IF _bIsFirstSeg AND _bIsLastSeg THEN	
	_sPath := '';
    _nLen := 0;
	_nSegStart := 0;
	_nSegEnd := 0;
	RemoveAndNext := Ok;
ELSIF _bIsFirstSeg THEN
	_sPath := Tc2_Standard.DELETE(_sPath, _nSegLen + 1, _nSegStart); // Also removes dot after first segment
	_nLen := _nLen - _nSegLen;
	_nSegStart := 0;
	_nSegEnd := 0;
	RemoveAndNext := Ok;
ELSIF _bIsLastSeg THEN
	_sPath := Tc2_Standard.DELETE(_sPath, _nSegLen + 1, _nSegStart - 1); // Also removes dot before last segment
	_nLen := _nLen - _nSegLen;
	_nSegStart := 0;
	_nSegEnd := 0;
	RemoveAndNext := Ok;
ELSE
	_sPath := Tc2_Standard.DELETE(_sPath, _nSegLen + 1, _nSegStart); // Also removes dot after segment
	_nLen := _nLen - _nSegLen;
	_nSegStart := _nSegEnd + 2; // Skip the delimiter
	
	FOR i := _nSegStart TO _nLen DO
		IF Tc2_Standard.MID(_sPath, 1, i) = '.' THEN
			_nSegEnd := i - 1;
			EXIT;
		END_IF;
	END_FOR;
	
	// If no more delimiters, this is the last segment
	IF _nSegEnd < _nSegStart THEN
		_nSegEnd := _nLen;
	END_IF;
	RemoveAndNext := Ok;
END_IF
END_METHOD

// Removes the current segment and moves to the previous segment.
// Returns `Ok` if successful, `None` if no segment to remove.
METHOD RemoveAndPrev : Result
VAR
    _nSegLen		: INT := _nSegEnd - _nSegStart + 1; // Length of the segment to remove
    _bIsFirstSeg	: BOOL := (_nSegStart = 1); // Check if the segment is the first segment
    _bIsLastSeg		: BOOL := (_nSegEnd = _nLen); // Check if the segment is the last segment
	i				: INT;
END_VAR
// Ensure the current path is valid
IF _sPath = '' OR _nSegStart = 0 THEN
    RemoveAndPrev := None;
    RETURN;
END_IF;

IF _bIsFirstSeg AND _bIsLastSeg THEN	
	_sPath := '';
    _nLen := 0;
	_nSegStart := 0;
	_nSegEnd := 0;
	RemoveAndPrev := Ok;
ELSIF _bIsFirstSeg THEN
	_sPath := Tc2_Standard.DELETE(_sPath, _nSegLen + 1, _nSegStart); // Also removes dot after first segment
	_nLen := _nLen - _nSegLen;
	_nSegStart := 0;
	_nSegEnd := 0;
	RemoveAndPrev := Ok;
ELSIF _bIsLastSeg THEN
	_sPath := Tc2_Standard.DELETE(_sPath, _nSegLen + 1, _nSegStart - 1); // Also removes dot before last segment
	_nLen := _nLen - _nSegLen;
	_nSegStart := 0;
	_nSegEnd := 0;
	RemoveAndPrev := Ok;
ELSE
	_sPath := Tc2_Standard.DELETE(_sPath, _nSegLen + 1, _nSegStart); // Also removes dot after segment
	_nLen := _nLen - _nSegLen;
	_nSegEnd := _nSegStart - 2; // Skip the delimiter
	
	FOR i := _nSegEnd TO 1 BY -1 DO
		IF Tc2_Standard.MID(_sPath, 1, i) = '.' THEN
			_nSegStart := i + 1;
			EXIT;
		END_IF;
	END_FOR;
	
	// If no more delimiters, this is the first segment
	IF _nSegEnd < _nSegStart THEN
		_nSegStart := 1;
	END_IF;
	RemoveAndPrev := Ok;
END_IF
END_METHOD

// Sets the symbolic path to a new value.
// Validates the input path for correctness.
// Returns `Ok` if successful, `None` if invalid.
METHOD Set : Result
VAR_INPUT
    sNewPath : Str; // New path to set
END_VAR

VAR
	i				: INT;
	_nStrLen		: INT := Tc2_Standard.LEN(sNewPath);
	_sChar			: Ch;
END_VAR
IF sNewPath = '' THEN
	Set := None;
	RETURN;
END_IF

_sChar := Tc2_Standard.MID(sNewPath, 1, 1);
IF (_sChar >= '0') AND (_sChar <= '9') THEN
	Set := None;
    RETURN;
END_IF;

sNewPath := Tc2_Utilities.F_ToLCase(sNewPath);

FOR i := 1 TO _nStrLen DO
    _sChar := Tc2_Standard.MID(sNewPath, 1, i);
    
    // Check for invalid characters
    IF NOT ((_sChar >= 'a' AND _sChar <= 'z') OR 	// Lowercase letters
            (_sChar >= '0' AND _sChar <= '9') OR 	// Numbers
            (_sChar = '_') OR                 		// Underscore
			(_sChar = '.') OR
			(_sChar = '*')) THEN					// Wildcard
		Set := None;
        RETURN;
    END_IF;
END_FOR;

IF Tc2_Standard.FIND(sNewPath, '..') <> 0 THEN
	Set := None;
	RETURN;
END_IF

IF Tc2_Standard.FIND(sNewPath, '**') <> 0 THEN
	Set := None;
	RETURN;
END_IF

_sPath := sNewPath;
_nLen := _nStrLen;
Set := Ok;
END_METHOD

// Replaces the current segment with a new segment.
// Returns `Ok` if successful, `None` if invalid.
METHOD Swap : Result
VAR_INPUT
    sToSwap : Str; // New segment to replace the current segment
END_VAR
VAR
	_nSegLen	: INT := _nSegEnd - _nSegStart + 1;
	_nSwapLen	: INT := Tc2_Standard.LEN(sToSwap);
	_nNewLen	: INT := _nLen - _nSegLen + _nSwapLen;
END_VAR
IF _sPath = '' OR _nSegStart = 0 OR sToSwap = '' THEN
    Swap := None;
    RETURN;
END_IF;

IF _HasIncorrectSymbols(sToSwap) THEN
	Swap := None;
	RETURN;
END_IF

IF _nNewLen <= 255 THEN
	_sPath := Tc2_Standard.REPLACE(_sPath, sToSwap, _nSegLen, _nSegStart);
	_nSegEnd := _nSegStart + _nSwapLen - 1;
	_nLen := _nNewLen;
	Swap := Ok;
END_IF
END_METHOD

END_FUNCTION_BLOCK

// Broadcast/Helpers/GetSignal
(*
Searches an `I_Entity` for a `I_Signal` component matching provided id pattern.
Result:
- Ok - Returns `I_Signal`.
- Err.NotFound - Returns null.
- Err.InvRef - Returns null.
- Err.Itf0 - Returns null, incorrect interface.
*)
FUNCTION GetSignal : Result
VAR_INPUT
	iEntity		: I_Entity;
	sTagId		: Str;
	iOut		: REFERENCE TO I_Signal;
END_VAR
VAR
	i			: Iter(1);
	_iComp		: I_FatComponent;
	cmp			: TagCmp;
END_VAR

IF iEntity = 0 THEN
	GetSignal := Err.Itf0;
	RETURN;
END_IF

IF NOT __ISVALIDREF(iOut) THEN
	GetSignal := Err.InvRef;
	RETURN;
END_IF

WHILE IsOk(iEntity.Get(i.Next(), _iComp)) DO
	IF IsOk(ICompToISignal(_iComp.Raw, iOut)) THEN
		IF cmp.Set(iOut.Tag).MatchWcdId(sTagId).IsTrue() THEN
			GetSignal := Ok;
			RETURN;
		ELSE
			iOut := 0;
		END_IF
	END_IF
END_WHILE

GetSignal := Err.NotFound;

END_FUNCTION

// Broadcast/Signal/ICompToISignal
(*
Casts I_Component as I_Signal.
Returns:
- Ok - Success,
- Err.InvRef - Invalid reference,
- Err.Itf0 - Invalid interface,
- Err.NoMatch - Cast failed
*)
FUNCTION ICompToISignal : Result
VAR_INPUT
	iIn	: I_Component;
	iOut: REFERENCE TO I_Signal;
END_VAR

IF NOT __ISVALIDREF(iOut) THEN
	ICompToISignal := Err.InvRef;
	RETURN;
END_IF

IF iIn = 0 THEN
	ICompToISignal := Err.Itf0;
	RETURN;
END_IF

IF __QUERYINTERFACE(iIn, iOut) THEN
	ICompToISignal := Ok;
ELSE
	ICompToISignal := Err.NoMatch;
END_IF

END_FUNCTION

// Broadcast/Receiver/AbstractReceiver
FUNCTION_BLOCK ABSTRACT AbstractReceiver IMPLEMENTS I_Callable, I_Receiver
VAR
	_tag: Tag;
END_VAR

(*
This method provides a standardized way for other objects to interact with the object that owns it.
*)
METHOD Call
VAR_INPUT
	iArg	: I_Arg;
END_VAR
END_METHOD

METHOD INTERNAL Receive
VAR_INPUT
	iArg			: I_Arg;
END_VAR
Call(iArg);
END_METHOD

(*
Provides access to the tag associated with the signal.
*)
PROPERTY FINAL Tag : I_Tag
GET
Tag := _tag;
END_GET
END_PROPERTY

END_FUNCTION_BLOCK

// Dbg/DebugInfo
(*
Provides access to registered debug information, enabling monitoring and troubleshooting of system components.
*)
FUNCTION_BLOCK DebugInfo
VAR
	_lastMsgIdx			: REFERENCE TO UDINT REF= _Debug.nLastMsg;
	_msg				: REFERENCE TO ARRAY[1..Param.DEBUGMSG_CAP] OF _DebugInfo REF= _Debug.debugMsg;
	
	_lastStrIdx			: REFERENCE TO UDINT REF= _Debug.nLastStr;
	_str				: REFERENCE TO ARRAY[1..Param.DEBUGSTR_CAP] OF Str REF= _Debug.debugStr;
END_VAR

END_FUNCTION_BLOCK

// Dbg/DebugStr
(*
Logs a debug message as a string without associating it with a specific component.
*)
FUNCTION DebugStr
VAR_INPUT
	sInfo			: Str;
END_VAR
VAR
END_VAR

IF _Debug.nLastStr < Param.DEBUGSTR_CAP THEN
	_Debug.nLastStr := _Debug.nLastStr + 1;
ELSE
	_Debug.nLastStr := 1;
END_IF

_Debug.debugStr[_Debug.nLastStr] := sInfo;

END_FUNCTION

// Entity/Core/Entity/EntityEnd
(*
Defines end of an entity scope outside which no new component can be registered.
*)
FUNCTION_BLOCK EntityEnd IMPLEMENTS I_Debug

//FB_Init is always available implicitly and it is used primarily for initialization.
//The return value is not evaluated. For a specific influence, you can also declare the
//methods explicitly and provide additional code there with the standard initialization
//code. You can evaluate the return value.
{attribute 'hide'}
METHOD FB_Init: BOOL
VAR_INPUT
    bInitRetains: BOOL; // TRUE: the retain variables are initialized (reset warm / reset cold)
    bInCopyCode: BOOL;  // TRUE: the instance will be copied to the copy code afterward (online change)   
END_VAR
VAR
	_nResult	: Result;
END_VAR
IF IsErr(_EndEntity(), nOut => _nResult) THEN
	DebugMsg(THIS^, Tc2_Standard.CONCAT('_EndEntity() failed with code: ', ResultToStr(_nResult)));
END_IF
END_METHOD

END_FUNCTION_BLOCK

// Entity/Sys/_Helpers/_EndEntity
FUNCTION INTERNAL _EndEntity : Result
VAR
	i						: UDINT;
END_VAR

IF NOT _Runtime.bInit THEN
	_EndEntity := Err.Init;
	RETURN;
END_IF

IF _Ec.iUnderConstruction = 0 THEN
	_EndEntity := Err.Itf0;
	RETURN;
END_IF

_Ec.iUnderConstruction._IsCompleted := TRUE;

_Ec.nConstructedScopes := _Ec.nConstructedScopes - 1;
IF _Ec.nConstructedScopes > 0 THEN
	FOR i := _Ec.nEntityLen TO 1 BY -1 DO
		IF NOT _Ec.iEntity[i]._IsCompleted THEN
			_Ec.iUnderConstruction := _Ec.iEntity[i];
			_EndEntity := Ok;
			RETURN;
		END_IF
	END_FOR
	
	// All completed
	_EndEntity := Ok;
ELSE
	_Ec.iUnderConstruction := 0;
	_EndEntity := Ok;
END_IF

END_FUNCTION

// Entity/Core/Entity/EntityExtend
(*
Reopens an entity scope for modifications.
*)
FUNCTION_BLOCK EntityExtend IMPLEMENTS I_Debug

//FB_Init is always available implicitly and it is used primarily for initialization.
//The return value is not evaluated. For a specific influence, you can also declare the
//methods explicitly and provide additional code there with the standard initialization
//code. You can evaluate the return value.
{attribute 'hide'}
METHOD FB_Init: BOOL
VAR_INPUT
    bInitRetains: BOOL; // TRUE: the retain variables are initialized (reset warm / reset cold)
    bInCopyCode: BOOL;  // TRUE: the instance will be copied to the copy code afterward (online change)
	
	iEntity	: I_EntityNode;
END_VAR
VAR
	_nResult	: Result;
END_VAR
IF IsErr(_ExtendEntity(iEntity), nOut => _nResult) THEN
	DebugMsg(THIS^, Tc2_Standard.CONCAT('_ExtendEntity(I_EntityNode) failed with code: ', ResultToStr(_nResult)));
END_IF
END_METHOD

END_FUNCTION_BLOCK

// Entity/Sys/_Helpers/_ExtendEntity
FUNCTION INTERNAL _ExtendEntity : Result
VAR_INPUT
	iEntity	: I_EntityNode;
END_VAR

IF NOT _Runtime.bInit THEN
	_ExtendEntity := Err.Init;
	RETURN;
END_IF

IF iEntity = 0 THEN
	_ExtendEntity := Err.Itf0;
	RETURN;
END_IF

iEntity._IsCompleted := FALSE;
_Ec.iUnderConstruction := iEntity;
_Ec.nConstructedScopes := _Ec.nConstructedScopes + 1;

_ExtendEntity := Ok;

END_FUNCTION

// Entity/Core/Entity/EntityStart
(*
Represents a registered entity in the Entity-Component system and start of its scope.
Nested scopes are possible, components are always registered within most inner scope.
*)
FUNCTION_BLOCK EntityStart IMPLEMENTS I_Entity, I_Debug;
VAR
	_nId		: UDINT;
	_nStart		: UDINT;
	_nEnd		: UDINT;
	_nSize		: UDINT;
	_bIsCompleted	: BOOL;
END_VAR

PROPERTY INTERNAL _AsIEntity : I_Entity
GET
_AsIEntity := THIS^;
END_GET
END_PROPERTY

PROPERTY INTERNAL _End : UDINT
GET
_End := _nEnd;
END_GET
SET
_nEnd := _End;
END_SET
END_PROPERTY

PROPERTY INTERNAL _IsCompleted : BOOL
GET
_IsCompleted := _bIsCompleted;
END_GET
SET
_bIsCompleted := _IsCompleted;
END_SET
END_PROPERTY

PROPERTY INTERNAL _Size : UDINT
GET
_Size := _nSize;
END_GET
SET
_nSize := _Size;
END_SET
END_PROPERTY

PROPERTY INTERNAL _Start : UDINT
GET
_Start := _nStart;
END_GET
SET
_nStart := _Start;
END_SET
END_PROPERTY

//FB_Init is always available implicitly and it is used primarily for initialization.
//The return value is not evaluated. For a specific influence, you can also declare the
//methods explicitly and provide additional code there with the standard initialization
//code. You can evaluate the return value.
{attribute 'hide'}
METHOD FB_Init: BOOL
VAR_INPUT
    bInitRetains: BOOL; // TRUE: the retain variables are initialized (reset warm / reset cold)
    bInCopyCode: BOOL;  // TRUE: the instance will be copied to the copy code afterward (online change)
END_VAR
VAR
	_nResult	: Result;
END_VAR
IF IsErr(_StartEntity(THIS^, nIndex => _nId), nOut => _nResult) THEN
	DebugMsg(THIS^, Tc2_Standard.CONCAT('_StartEntity(THIS^) failed with code: ', ResultToStr(_nResult)));
END_IF
END_METHOD

(*
Retrieves a specific component from the entity based on the provided index.  
Returns `Err.NotFound` if the index is out of range or the entity size is zero.
Returns `Err.InvRef` if the reference to interface variable is invalid.
Otherwise returns `Ok`.
*)
METHOD Get : Result
VAR_INPUT
	nIndex	: UDINT;
	iOut	: REFERENCE TO I_FatComponent;
END_VAR
IF NOT __ISVALIDREF(iOut) THEN
	Get := Err.InvRef;
	RETURN;
END_IF

IF nIndex > _nSize - 1 OR_ELSE nIndex = 0 OR_ELSE _nSize = 0 THEN
	Get := Err.NotFound;
	RETURN;
END_IF

iOut := _Ec.comp[_nStart + nIndex].variant.iComponent;
Get := Ok;
END_METHOD

(*
Returns the unique identifier of the entity, used for tracking and referencing within the EC system.
*)
PROPERTY Id : UDINT
GET
Id := _nId;
END_GET
END_PROPERTY

(*
Provides the size of the entity, indicating the number of components it manages.  
Note: For internal logic purposes, this value is incremented by one beyond the actual component count.
*)
PROPERTY Size : UDINT
GET
Size := _nSize;
END_GET
END_PROPERTY

END_FUNCTION_BLOCK

// Entity/Sys/_Helpers/_StartEntity
// ---------------------------------------------------------------------------
// FUNCTION:  _RegEntity
// PURPOSE:   Registers (adds) a new entity into the global _Ec.iEntity array.
//            Increments nEntityLen, assigns the entity to the next free index,
//            and sets the entity's Id to that index.
//
// NOTE:
//   - Fails if iEntity = 0 (null pointer) or if the array is at max capacity.
// ---------------------------------------------------------------------------
FUNCTION INTERNAL _StartEntity : Result
VAR_INPUT
    iEntity : I_EntityNode;
END_VAR
VAR_OUTPUT
    nIndex  : UDINT;
END_VAR

IF NOT _Runtime.bInit THEN
	_StartEntity := Err.Init;
	RETURN;
END_IF

IF iEntity = 0 THEN
	_StartEntity := Err.Itf0;
	RETURN;
END_IF

IF _Ec.nEntityLen = Param.ENTITY_CAP THEN
	_StartEntity := Err.Ovf;
	RETURN;
END_IF

_Ec.nEntityLen := _Ec.nEntityLen + 1;
_Ec.iEntity[_Ec.nEntityLen] := iEntity;
nIndex := _Ec.nEntityLen;

_Ec.iUnderConstruction := iEntity;
_Ec.nConstructedScopes := _Ec.nConstructedScopes + 1;

_StartEntity := Ok;

END_FUNCTION

// Entity/Core/GetEntity
(*
Retrieves the I_Entity instance at the given nIndex from the global entity list.
Returns:
- Ok - Returns I_Entity
- Err.NotFound - Returns Null
- Err.InvRef - Returns Null, invalid reference
*)
FUNCTION GetEntity : Result
VAR_INPUT
	nIndex		: UDINT;
	iOut		: REFERENCE TO I_Entity;
END_VAR

IF NOT __ISVALIDREF(iOut) THEN
	GetEntity := Err.InvRef;
	RETURN;
END_IF

IF nIndex > _Ec.nEntityLen OR nIndex = 0 THEN
	GetEntity := Err.NotFound;
	RETURN;
END_IF

iOut := _Ec.iEntity[nIndex]._AsIEntity;
GetEntity := Ok;

END_FUNCTION

// Entity/Core/GetOwnerFromRaw
(*
Finds the owning entity of a given component in the Entity-Component system.  
This function may involve a costly search operation, iterating through all components.
Returns:
- `Ok` - Successfully retrieves the `I_Entity` that owns the component.
- `Err.Itf0` - iIn = 0.
- `Err.InvRef` - Invalid output reference.
- `Err.NotFound` - No owning entity is found, returning null.
*)
FUNCTION GetOwnerFromRaw : Result
VAR_INPUT
	iIn: I_Component;
	iOut: REFERENCE TO I_Entity;
END_VAR
VAR
	i			: Iter(1);
	j			: Iter(1);
	_iComp		: I_FatComponent;
END_VAR

IF iIn = 0 THEN
	GetOwnerFromRaw := Err.Itf0;
	RETURN;
END_IF

IF NOT __ISVALIDREF(iOut) THEN
	GetOwnerFromRaw := Err.InvRef;
	RETURN;
END_IF

WHILE IsOk(GetEntity(i.Next(), iOut)) DO
	j.Set(1);
	WHILE IsOk(iOut.Get(j.Next(), _iComp)) DO
		IF _iComp.Raw = iIn THEN
			GetOwnerFromRaw := Ok;
			RETURN;
		END_IF
	END_WHILE
END_WHILE

GetOwnerFromRaw := Err.NotFound;

END_FUNCTION

// Entity/List/CompList
(*
A list implementation for managing `I_Arg`.  
*)
FUNCTION_BLOCK CompList
VAR_GENERIC CONSTANT
	nCap	: UDINT := 100;
END_VAR

IMPLEMENTS I_MutCompList

VAR
	_iList	: ARRAY[1..nCap] OF I_Component;
END_VAR

(*
Provides the maximum capacity of the list.
*)
PROPERTY Cap : UDINT
GET
Cap := nCap;
END_GET
END_PROPERTY

(*
Retrieves the `I_Component` at the specified index.  
Returns:
- `Ok` - Successfully retrieves the `I_Component`.
- `Err.Idx` - The specified index is out of bounds.
- `Err.InvRef` - Invalid output reference.
- `Err.Idx` - `iOut` = 0.
*)
METHOD Get : Result
VAR_INPUT
	nIndex		: UDINT;
	iOut		: REFERENCE TO I_Component;
END_VAR
IF nIndex > nCap OR nIndex = 0 THEN
	Get := Err.Idx;
	RETURN;	
END_IF

IF NOT __ISVALIDREF(iOut) THEN
	Get := Err.InvRef;
	RETURN;
END_IF

iOut := _iList[nIndex];
IF iOut <> 0 THEN
	Get := Ok;
ELSE
	Get := Err.NotFound;
END_IF
END_METHOD

(*
Adds, updates, or removes an argument in the list at the specified index.  
Return:
- `Ok` - Upon successfully adding, modifying, or removing an entry.
- `Err.Idx` - When attempting to modify an entry at an out-of-bounds index.
*)
METHOD Set : Result
VAR_INPUT
	iIn			: I_Component;
	nIndex		: UDINT;
END_VAR
IF nIndex > nCap OR nIndex = 0 THEN
	Set := Err.Idx;
	RETURN;	
END_IF

_iList[nIndex] := iIn;
Set := Ok;
END_METHOD

END_FUNCTION_BLOCK

// Entity/List/I_MutCompList
(*
A list implementation for managing `I_Component`.  
*)
INTERFACE I_MutCompList EXTENDS I_CompList

(*
Adds, updates, or removes an argument in the list at the specified index.  
Return:
- `Ok` - Upon successfully adding, modifying, or removing an entry.
- `Err.Idx` - When attempting to modify an entry at an out-of-bounds index.
*)
METHOD Set : Result
VAR_INPUT
	iIn			: I_Component;
	nIndex		: UDINT;
END_VAR
END_METHOD

END_INTERFACE

// Entity/List/I_CompList
(*
A list implementation for managing `I_Component`.  
*)
INTERFACE I_CompList EXTENDS I_Debug

(*
Provides the maximum capacity of the list.
*)
PROPERTY Cap : UDINT
GET
END_GET
END_PROPERTY

(*
Retrieves the `I_Component` at the specified index.  
Returns:
- `Ok` - Successfully retrieves the `I_Component`.
- `Err.Idx` - The specified index is out of bounds.
- `Err.InvRef` - Invalid output reference.
- `Err.Idx` - `iOut` = 0.
*)
METHOD Get : Result
VAR_INPUT
	nIndex		: UDINT;
	iOut		: REFERENCE TO I_Component;
END_VAR
END_METHOD

END_INTERFACE

// Entity/Set/CompSet
FUNCTION_BLOCK CompSet

VAR_GENERIC CONSTANT
	CAP: UDINT := 10;
END_VAR

IMPLEMENTS I_CompSet

VAR_OUTPUT
END_VAR
VAR
	_iComp: ARRAY[1..CAP] OF I_Component;
	_nLen: UDINT;
END_VAR

METHOD Append : Result
VAR_INPUT
	iComp: I_Component;
END_VAR
IF _nLen = CAP THEN
	Append := Err.Ovf;
	RETURN;
END_IF

IF iComp = 0 THEN
	Append := Err.Itf0;
	RETURN;
END_IF

_nLen := _nLen + 1;
_iComp[_nLen] := iComp;
Append := Ok;
END_METHOD

METHOD Get : Result
VAR_INPUT
	nIdx: UDINT;
	iResult: REFERENCE TO I_Component;
END_VAR
IF nIdx = 0 OR nIdx > CAP THEN
	Get := Err.Ovf;
	RETURN;
END_IF

IF NOT __ISVALIDREF(iResult) THEN
	Get := Err.InvRef;
	RETURN;
END_IF

iResult := _iComp[nIdx];
Get := Ok;
END_METHOD

END_FUNCTION_BLOCK

// Entity/Set/I_CompSet
INTERFACE I_CompSet

METHOD Append : Result
VAR_INPUT
	iComp: I_Component;
END_VAR
END_METHOD

METHOD Get : Result
VAR_INPUT
	nIdx: UDINT;
	iResult: REFERENCE TO I_Component;
END_VAR
END_METHOD

END_INTERFACE

// Result/IsFail
// Return TRUE on a NON successful (NOT Ok) result.
// Optionally carries the value over to nOut for further processing.
FUNCTION IsFail : BOOL
VAR_INPUT
    nIn : Result; // Result variable to check for success
END_VAR
VAR_OUTPUT
    nOut : Result; // Carries the input value for further use
END_VAR

IsFail := nIn <= 0;
nOut := nIn;

END_FUNCTION

// Runtime/Execute/Execute
(*
Allows registration of FB implementing `I_Execute`. 
*)
FUNCTION_BLOCK FINAL Execute IMPLEMENTS I_ExecuteNode, I_Debug
VAR
	_iExecute		: I_Execute;
	_iNext			: I_ExecuteNode;
	_nState			: Result;
	_nPhase			: INT;
END_VAR

METHOD INTERNAL Attach : Result
VAR_INPUT
	iExecute		: I_ExecuteNode;
END_VAR
VAR
	_iThis			: I_ExecuteNode := THIS^;
END_VAR
IF iExecute = 0 THEN
	DebugMsg(0, Tc2_Standard.CONCAT(__POUNAME(), ': Itf = 0!'));
	RETURN;
END_IF

IF _iThis <> _Runtime.iLastCyclic THEN
	DebugMsg(THIS^, Tc2_Standard.CONCAT(__POUNAME(), ': Is not the last node!'));
	RETURN;
END_IF

IF IsSome(iExecute.state) THEN
	DebugMsg(iExecute, Tc2_Standard.CONCAT(__POUNAME(), ': Has already been added!'));
	RETURN;
END_IF

_Runtime.iLastCyclic := iExecute;
_iNext := iExecute;
END_METHOD

METHOD INTERNAL Exe
VAR_INPUT
END_VAR
_iExecute.Execute(_nPhase);

IF _iNext <> 0 THEN
	_iNext.Exe();
END_IF
END_METHOD

//FB_Init is always available implicitly and it is used primarily for initialization.
//The return value is not evaluated. For a specific influence, you can also declare the
//methods explicitly and provide additional code there with the standard initialization
//code. You can evaluate the return value.
{attribute 'hide'}
METHOD FB_Init: BOOL
VAR_INPUT
    bInitRetains: BOOL; // TRUE: the retain variables are initialized (reset warm / reset cold)
    bInCopyCode: BOOL;  // TRUE: the instance will be copied to the copy code afterward (online change)
	
	iExecute			: I_Execute;
END_VAR
IF IsSome(_nState) THEN
	RETURN;
END_IF

IF (_iExecute := iExecute) = 0 THEN
	_nState := Err.Itf0;
	DebugMsg(THIS^, Tc2_Standard.CONCAT(__POUNAME(), ': Itf = 0!'));
	RETURN;
END_IF



IF _Runtime.iLastCyclic <> 0 THEN
	IF IsErr(_Runtime.iLastCyclic.Attach(THIS^), nOut => _nState) THEN
		DebugMsg(THIS^, Tc2_Standard.CONCAT(__POUNAME(), ': Error Inside!'));
	END_IF
ELSE
	_Runtime.iFirstCyclic := THIS^;
	_Runtime.iLastCyclic := THIS^;
	_nState := Ok;
END_IF
END_METHOD

PROPERTY Phase : INT
GET
Phase := _nPhase;
END_GET
SET
_nPhase := Phase;
END_SET
END_PROPERTY

PROPERTY INTERNAL State : Result
GET
State := _nState;
END_GET
SET
IF IsNone(_nState) THEN
	_nState := State;
END_IF
END_SET
END_PROPERTY

END_FUNCTION_BLOCK

// Runtime/Execute/I_Execute
(*
A `Execute` method of FB implmenting this interface will be called every control loop cycle.
*)
INTERFACE I_Execute EXTENDS I_Debug

(*
If registered, this method will be executed cyclically.
*)
METHOD Execute
VAR_INPUT
	nPhase: INT;
END_VAR
END_METHOD

END_INTERFACE

// Runtime/Execute/I_ExecuteNode
INTERFACE INTERNAL I_ExecuteNode EXTENDS I_Debug;

METHOD INTERNAL Attach : Result
VAR_INPUT
	iExecute		: I_ExecuteNode;
END_VAR
END_METHOD

METHOD INTERNAL Exe
VAR_INPUT
END_VAR
END_METHOD

PROPERTY INTERNAL State : Result
GET
END_GET
SET
END_SET
END_PROPERTY

END_INTERFACE

// Runtime/Runtime
(*
Manages the initialization and cyclic execution of registered function blocks.
*)
FUNCTION Runtime

IF _Runtime.bInit THEN
	IF _Runtime.iFirstInit <> 0 THEN
		_Runtime.iFirstInit.Init();
	END_IF
	_Runtime.bInit := FALSE;

	IF _Ec.nConstructedScopes <> 0 THEN
		DebugMsg(0, 'Close all Entity scopes!');
	END_IF
	
	IF _Debug.nErrorNumber > 0 THEN
		_Runtime.iFirstCyclic := 0;
		Tc2_System.ADSLOGSTR(Tc2_System.ADSLOG_MSGTYPE_ERROR, Tc2_Standard.CONCAT('Runtime disabled! Errors: ', UDINT_TO_STRING(_Debug.nErrorNumber)), '');
	END_IF
END_IF

IF _Runtime.iFirstCyclic <> 0 THEN
	_Runtime.iFirstCyclic.Exe();
END_IF

END_FUNCTION

// State/_Buffer/_StateBuffer
(*
A buffer for storing states.  
*)
FUNCTION_BLOCK INTERNAL _StateBuffer
VAR
	_iFirst				: I_StateInternal;
	_iLast				: I_StateInternal;
	_nLen				: UDINT;
END_VAR

(*
Returns the current number of states stored in the buffer.
*)
METHOD Length : UDINT
VAR_INPUT
END_VAR
Length := _nLen;
END_METHOD

(*
Removes and retrieves the oldest state from the buffer.  

Returns:
- `Ok` - If a state is successfully removed.
- `None` - If the buffer is empty.
*)
METHOD Pop : Result
VAR_OUTPUT
	iState			: I_StateInternal;
END_VAR
IF _iFirst = 0 THEN
	Pop := None;
	RETURN;
END_IF

iState := _iFirst;
_iFirst := _iFirst._NextInBuffer;
iState._NextInBuffer := 0;
iState._InQueue := FALSE;

IF _iFirst = 0 THEN
	_iLast := 0;
END_IF

_nLen := _nLen - 1;
Pop := Ok;
END_METHOD

(*
Adds a new state to the buffer.  
Returns:
- `Ok` - If the state is successfully added.
- `Err.Itf0` - If the provided state interface is invalid.
- `Err.IncArg` - Uf the provided state already is in some buffer.
*)
METHOD Push : Result
VAR_INPUT
	iState			: I_StateInternal;
END_VAR
IF iState = 0 THEN
	Push := Err.Itf0;
	RETURN;
END_IF

IF iState._InQueue THEN
	Push := Err.IncArg;
	RETURN;
END_IF

IF _iLast = 0 THEN
	_iFirst := iState;
	_iLast := iState;
	iState._InQueue := TRUE;
	_nLen := _nLen + 1;
ELSE
	_iLast._NextInBuffer := iState;
	_iLast := iState;
	iState._InQueue := TRUE;
	_nLen := _nLen + 1;
END_IF

Push := Ok;
END_METHOD

END_FUNCTION_BLOCK

// State/_Machine/_StateMachine
FUNCTION_BLOCK INTERNAL _StateMachine IMPLEMENTS I_Execute
VAR
	_exe					: Execute(THIS^);
	_iCurrentState			: I_StateInternal;
END_VAR

(*
Changes the current state to a new state.  

Returns:
- `Ok` - If the state transition is successful.
- `Err.Itf0` - If the new state interface is invalid.
- `None` - If the transition cannot be completed due to state conditions.
*)
METHOD Change : Result
VAR_INPUT
	iNewState	: I_StateInternal;
END_VAR
VAR_OUTPUT
	iOldState	: I_StateInternal;
END_VAR
IF iNewState = 0 THEN
	Change := Err.Itf0;
	RETURN;
END_IF

IF iNewState = _iCurrentState THEN
	Change := None;
	RETURN;
END_IF

IF NOT iNewState._CanActivate() THEN
	Change := None;
	RETURN;
END_IF

IF _iCurrentState <> 0 AND_THEN NOT _iCurrentState._CanDeactivate() THEN
	Change := None;
	RETURN;
END_IF

IF _iCurrentState <> 0 THEN
	_iCurrentState._OnExit();
END_IF

iNewState._OnEntry();
iOldState := _iCurrentState;
_iCurrentState := iNewState;
Change := Ok;
END_METHOD

METHOD Execute
VAR_INPUT
	nPhase: INT := 0;
END_VAR
IF _iCurrentState <> 0 THEN
	_iCurrentState._OnExecute();
END_IF
END_METHOD

(*
Provides access to the current state, enabling inspection or external interaction with the state.
*)
PROPERTY State : I_State
GET
State := _iCurrentState._AsIState;
END_GET
END_PROPERTY

END_FUNCTION_BLOCK

// State/Helpers/GetState
(*
Searches an `I_Entity` for a `I_State` component matching provided id pattern.
Result:
- Ok - Returns `I_State`.
- Err.NotFound - Returns null.
- Err.InvRef - Returns null.
- Err.Itf0 - Returns null, incorrect interface.
*)
FUNCTION GetState : Result
VAR_INPUT
	iEntity		: I_Entity;
	sTagId		: Str;
	iOut		: REFERENCE TO I_State;
END_VAR
VAR
	i			: Iter(1);
	_iComp		: I_FatComponent;
	cmp			: TagCmp;
END_VAR

IF iEntity = 0 THEN
	GetState := Err.Itf0;
	RETURN;
END_IF

IF NOT __ISVALIDREF(iOut) THEN
	GetState := Err.InvRef;
	RETURN;
END_IF

WHILE IsOk(iEntity.Get(i.Next(), _iComp)) DO
	IF IsOk(ICompToIState(_iComp.Raw, iOut)) THEN
		IF cmp.Set(iOut.Tag).MatchWcdId(sTagId).IsTrue() THEN
			GetState := Ok;
			RETURN;
		ELSE
			iOut := 0;
		END_IF
	END_IF
END_WHILE

GetState := Err.NotFound;

END_FUNCTION

// State/State/ICompToIState
(*
Casts I_Component as I_State.
Returns:
- Ok - Success,
- Err.InvRef - Invalid reference,
- Err.Itf0 - Invalid interface,
- Err.NoMatch - Cast failed
*)
FUNCTION ICompToIState : Result
VAR_INPUT
	iIn		: I_Component;
	iOut	: REFERENCE TO I_State;
END_VAR

IF NOT __ISVALIDREF(iOut) THEN
	ICompToIState := Err.InvRef;
	RETURN;
END_IF

IF iIn = 0 THEN
	ICompToIState := Err.Itf0;
	RETURN;
END_IF

IF __QUERYINTERFACE(iIn, iOut) THEN
	ICompToIState := Ok;
ELSE
	ICompToIState := Err.NoMatch;
END_IF

END_FUNCTION

// State/Helpers/GetStateManager
(*
Searches an `I_Entity` for a `I_StateManager` component matching provided id pattern.
Result:
- Ok - Returns `I_StateManager`.
- Err.NotFound - Returns null.
- Err.InvRef - Returns null.
- Err.Itf0 - Returns null, incorrect interface.
*)
FUNCTION GetStateManager : Result
VAR_INPUT
	iEntity		: I_Entity;
	iOut		: REFERENCE TO I_StateManager;
END_VAR
VAR
	i			: Iter(1);
	_iComp		: I_FatComponent;
	cmp			: TagCmp;
END_VAR

IF iEntity = 0 THEN
	GetStateManager := Err.Itf0;
	RETURN;
END_IF

IF NOT __ISVALIDREF(iOut) THEN
	GetStateManager := Err.InvRef;
	RETURN;
END_IF

WHILE IsOk(iEntity.Get(i.Next(), _iComp)) DO
	IF IsOk(ICompToIStateMgr(_iComp.Raw, iOut)) THEN
		GetStateManager := Ok;
		RETURN;
	END_IF
END_WHILE

GetStateManager := Err.NotFound;

END_FUNCTION

// State/Manager/ICompToIStateMgr
(*
Casts I_Component as I_StateManager.
Returns:
- Ok - Success,
- Err.InvRef - Invalid reference,
- Err.Itf0 - Invalid interface,
- Err.NoMatch - Cast failed
*)
FUNCTION ICompToIStateMgr : Result
VAR_INPUT
	iIn		: I_Component;
	iOut	: REFERENCE TO I_StateManager;
END_VAR

IF NOT __ISVALIDREF(iOut) THEN
	ICompToIStateMgr := Err.InvRef;
	RETURN;
END_IF

IF iIn = 0 THEN
	ICompToIStateMgr := Err.Itf0;
	RETURN;
END_IF

IF __QUERYINTERFACE(iIn, iOut) THEN
	ICompToIStateMgr := Ok;
ELSE
	ICompToIStateMgr := Err.NoMatch;
END_IF

END_FUNCTION

// State/Manager/I_StateManager
(*
Can be casted to `I_Component`.
Manages the lifecycle and transitions of states within an entity.  
Supports queuing state change requests, triggering state transitions, and broadcasting state change events.  
Adds a `_stateChangeEvent` Signal to the owning `I_Entity` during initialization, enabling external components to listen for state changes.
*)
INTERFACE I_StateManager EXTENDS I_Debug, I_Component

(*
Returns the entity that owns this state.
*)
PROPERTY Owner : I_Entity
GET
END_GET
END_PROPERTY

(*
Queues a request to transition to a specified state.  

Returns:
- `Ok` - If the state change request is successfully queued.
- `Err.Itf0` - If the provided state interface is invalid.
- `Err.NoMatch` - If the state does not belong to the same entity.
- `Err.IncArg` - If the state is already in the queue.
*)
METHOD Request : Result
VAR_INPUT
	iState		: I_State;
END_VAR
END_METHOD

(*
Retrieves the currently active state managed by the state manager.
*)
PROPERTY Current : I_State
GET
END_GET
END_PROPERTY

(*
Retrieves the state that is queued to become active next, but has not yet transitioned.
*)
PROPERTY Pretender : I_State
GET
END_GET
END_PROPERTY

(*
Retrieves the last active state prior to the current one.
*)
PROPERTY Previous : I_State
GET
END_GET
END_PROPERTY

END_INTERFACE

// State/Manager/StateManager
(*
Manages the lifecycle and transitions of states within an entity.  
Supports queuing state change requests, triggering state transitions, and broadcasting state change events.  
Adds a `_stateChangeEvent` Signal to the owning `I_Entity` during initialization, enabling external components to listen for state changes.
*)
FUNCTION_BLOCK FINAL StateManager IMPLEMENTS I_Execute, I_StateManager, I_Debug

VAR
	_comp				: Component(THIS^);

	_exe				: Execute(THIS^);
	_sm					: _StateMachine;
	_buffer				: _StateBuffer;
	
	_stateChangeEvent	: Signal;
	
	_iPretender			: I_State;
	_iCurrent			: I_State;
	_iPrevious 			: I_State;
	
	
END_VAR

// DO NOT CALL MANUALLY
{attribute 'hide'}
METHOD Execute
VAR_INPUT
	nPhase: INT := 0;
END_VAR
VAR
	_iNewState		: I_StateInternal;
	_iOldState		: I_StateInternal;
END_VAR
IF IsOk(_buffer.Pop(iState => _iNewState)) THEN
	_iPretender := _iNewState._AsIState;
	IF IsOk(_sm.Change(_iNewState, iOldState => _iOldState)) THEN
		_stateChangeEvent.Emit(_iNewState._AsIState.Tag);
		
		_iCurrent		:= _iNewState._AsIState;
		IF _iOldState <> 0 THEN
			_iPrevious		:= _iOldState._AsIState;
		END_IF
		
	END_IF
	
	_iPretender		:= 0;
END_IF
END_METHOD

(*
Returns the entity that owns this state.
*)
PROPERTY Owner : I_Entity
GET
Owner := _comp.Entity;
END_GET
END_PROPERTY

(*
Allows initializing an external interface variable with an interface pointer to this instance within declaration block.
Example:
iSMgr: I_StateManager;
smgr: StateManager := (Proxy := iSMgr);
Result: iSMgr <> 0 
*)
PROPERTY Proxy : REFERENCE TO I_StateManager
SET
Proxy := THIS^;
END_SET
END_PROPERTY

(*
Queues a request to transition to a specified state.  
Returns:
- `Ok` - If the state change request is successfully queued.
- `Err.Itf0` - If the provided state interface is invalid.
- `Err.NoMatch` - If the state does not belong to the same entity.
- `Err.IncArg` - If the state is already in the queue.
*)
METHOD Request : Result
VAR_INPUT
	iState			: I_State;
END_VAR
VAR
	iStateInternal	: I_StateInternal;
END_VAR
IF iState = 0 THEN
	Request := Err.Itf0;
	RETURN;
END_IF

IF iState.Owner <> _comp.Entity THEN
	Request := Err.NoMatch;
	RETURN;
END_IF

Request := _buffer.Push(iState._AsIStateInternal);
END_METHOD

(*
Retrieves the currently active state managed by the state manager.
*)
PROPERTY Current : I_State
GET
Current := _iCurrent;
END_GET
END_PROPERTY

(*
Retrieves the state that is queued to become active next, but has not yet transitioned.
*)
PROPERTY Pretender : I_State
GET
Pretender := _iPretender;
END_GET
END_PROPERTY

(*
Retrieves the last active state prior to the current one.
*)
PROPERTY Previous : I_State
GET
Previous := _iPrevious;
END_GET
END_PROPERTY

END_FUNCTION_BLOCK

// Strings/Strb/I_Strb
// A string builder utility that allows for manipulation of a string up to 255 characters. It implements the I_Strb interface that allows for method chaining.
INTERFACE INTERNAL I_Strb

// Appends the specified string to the current string.
// Truncates if the total length exceeds 255 characters.
METHOD Append : I_Strb
VAR_INPUT
    sToAdd : Str; // String to append
END_VAR
END_METHOD

// Finds the first occurrence of a substring after the specified position.
// Outputs the start and end positions of the found substring.
METHOD FindFirstAfter : I_Strb
VAR_INPUT
    sToFind : Str;      // Substring to find
    nPosition : INT := 1; // Starting position for search
END_VAR
VAR_OUTPUT
    nStart : INT;       // Start position of the found substring
    nEnd : INT;         // End position of the found substring
END_VAR
END_METHOD

// Finds the last occurrence of a substring before the specified position.
// Outputs the start and end positions of the found substring.
METHOD FindLastBefore : I_Strb
VAR_INPUT
    sToFind : Str;        // Substring to find
    nPosition : INT := 256; // Starting position for reverse search
END_VAR
VAR_OUTPUT
    nStart : INT;         // Start position of the found substring
    nEnd : INT;           // End position of the found substring
END_VAR
END_METHOD

// Checks if the specified substring exists after the given position.
METHOD HasAfter : BOOL
VAR_INPUT
    sToFind : Str;      // Substring to search for
    nPosition : INT := 0; // Starting position for search
END_VAR
VAR_OUTPUT
    nStart : INT;       // Start position of the found substring
    nEnd : INT;         // End position of the found substring
END_VAR
END_METHOD

// Checks if the specified substring exists before the given position.
METHOD HasBefore : BOOL
VAR_INPUT
    sToFind : Str;        // Substring to search for
    nPosition : INT := 256; // Ending position for reverse search
END_VAR
VAR_OUTPUT
    nStart : INT;         // Start position of the found substring
    nEnd : INT;           // End position of the found substring
END_VAR
END_METHOD

// Inserts a specified substring at a given position.
// Truncates if the total length exceeds 255 characters.
METHOD Inject : I_Strb
VAR_INPUT
    nPosition : INT;    // Position to inject the string
    sToInject : Str;    // String to inject
END_VAR
END_METHOD

// Checks if the current string is empty.
METHOD IsEmpty : BOOL
VAR_INPUT
END_VAR
END_METHOD

// Returns the current length of the string.
METHOD Length : INT
VAR_INPUT
END_VAR
END_METHOD

// Prepends the specified string to the current string.
// Truncates if the total length exceeds 255 characters.
METHOD Prepend : I_Strb
VAR_INPUT
    sToAdd : Str; // String to prepend
END_VAR
END_METHOD

// Returns the current string value.
METHOD Read : Str
VAR_INPUT
END_VAR
END_METHOD

// Removes a substring of specified length starting at a given position.
METHOD Remove : I_Strb
VAR_INPUT
    nLength : INT;    // Length of the substring to remove
    nPosition : INT;  // Starting position of the substring to remove
END_VAR
END_METHOD

// Sets the current string to a new value.
METHOD Set : I_Strb
VAR_INPUT
    sLiteral : Str; // New string value
END_VAR
END_METHOD

// Extracts a substring starting from a given position with a specified length.
METHOD Slice : I_Strb
VAR_INPUT
	nLength : INT;   // Length of the slice
    nPosition : INT; // Starting position of the slice
END_VAR
VAR_OUTPUT
    sSlice : Strb;   // The sliced string
END_VAR
END_METHOD

// Splits the string into two parts at the specified position.
METHOD Split : I_Strb
VAR_INPUT
    nPosition : INT; // Position to split the string
END_VAR
VAR_OUTPUT
    sLeft : Strb;    // Left part of the split
    sRight : Strb;   // Right part of the split
END_VAR
END_METHOD

END_INTERFACE

// Strings/Strb/Strb
// A string builder utility that allows for manipulation of a string up to 255 characters. It implements the I_Strb interface that allows for method chaining.
FUNCTION_BLOCK FINAL Strb IMPLEMENTS I_Strb
VAR
	_sString	: Str;
	_nLength	: INT;
END_VAR

PROPERTY PRIVATE _this : I_Strb
GET
VAR
	_iThis : I_Strb := THIS^;
END_VAR
_this := _iThis;
END_GET
END_PROPERTY

// Appends the specified string to the current string.
// Truncates if the total length exceeds 255 characters.
METHOD Append : I_Strb
VAR_INPUT
    sToAdd : Str; // String to append
END_VAR

VAR
	_nNewLength	: INT;
END_VAR
Append := _this;

IF sToAdd = '' THEN
	RETURN;
END_IF

_nNewLength := Tc2_Standard.LEN(sToAdd) + _nLength;
IF _nNewLength > 255 THEN
	_nNewLength := 255;
END_IF

_sString := Tc2_Standard.CONCAT(_sString, sToAdd);
_nLength := _nNewLength;
END_METHOD

// Finds the first occurrence of a substring after the specified position.
// Outputs the start and end positions of the found substring.
METHOD FindFirstAfter : I_Strb
VAR_INPUT
    sToFind : Str;      // Substring to find
    nPosition : INT := 1; // Starting position for search
END_VAR
VAR_OUTPUT
    nStart : INT;       // Start position of the found substring
    nEnd : INT;         // End position of the found substring
END_VAR

VAR
	_sTemp			: Str;
	_nOffset		: INT;
END_VAR
FindFirstAfter := _this;

IF sToFind = '' THEN
	RETURN;
END_IF

IF nPosition = 0 THEN
	RETURN;
END_IF

_sTemp := Tc2_Standard.MID(_sString, _nLength, nPosition);
IF (_nOffset := Tc2_Standard.FIND(_sTemp, sToFind)) <> 0 THEN
	nStart := nPosition + _nOffset - 1;
	nEnd := nPosition + _nOffset - 2 + Tc2_Standard.LEN(sToFind);
END_IF
END_METHOD

// Finds the last occurrence of a substring before the specified position.
// Outputs the start and end positions of the found substring.
METHOD FindLastBefore : I_Strb
VAR_INPUT
    sToFind : Str;        // Substring to find
    nPosition : INT := 256; // Starting position for reverse search
END_VAR
VAR_OUTPUT
    nStart : INT;         // Start position of the found substring
    nEnd : INT;           // End position of the found substring
END_VAR
VAR
	_sTemp			: Str;
	_nFindLength	: INT := Tc2_Standard.LEN(sToFind);
	_nOffset		: INT;
END_VAR
FindLastBefore := _this;

IF sToFind = '' THEN
	RETURN;
END_IF

IF nPosition = 0 THEN
	RETURN;
END_IF

IF nPosition = 256 THEN
	nPosition := _nLength;
END_IF

REPEAT
	_sTemp := Tc2_Standard.MID(_sString, _nFindLength, nPosition);
	IF _sTemp = sToFind THEN
		nStart 	:= nPosition;
		nEnd	:= nPosition + _nFindLength - 1;
		RETURN;
	END_IF
UNTIL
	(nPosition := nPosition - 1) <= 0
END_REPEAT
END_METHOD

// Checks if the specified substring exists after the given position.
METHOD HasAfter : BOOL
VAR_INPUT
    sToFind : Str;      // Substring to search for
    nPosition : INT := 0; // Starting position for search
END_VAR
VAR_OUTPUT
    nStart : INT;       // Start position of the found substring
    nEnd : INT;         // End position of the found substring
END_VAR
FindFirstAfter(sToFind, nPosition, nStart => nStart, nEnd => nEnd);
HasAfter := nStart > 0;
END_METHOD

// Checks if the specified substring exists before the given position.
METHOD HasBefore : BOOL
VAR_INPUT
    sToFind : Str;        // Substring to search for
    nPosition : INT := 256; // Ending position for reverse search
END_VAR
VAR_OUTPUT
    nStart : INT;         // Start position of the found substring
    nEnd : INT;           // End position of the found substring
END_VAR
IF nPosition = 256 THEN
	nPosition := Tc2_Standard.LEN(_sString);
END_IF

FindLastBefore(sToFind, nPosition, nStart => nStart, nEnd => nEnd);
HasBefore := nStart > 0;
END_METHOD

// Inserts a specified substring at a given position.
// Truncates if the total length exceeds 255 characters.
METHOD Inject : I_Strb
VAR_INPUT
    nPosition : INT;    // Position to inject the string
    sToInject : Str;    // String to inject
END_VAR
VAR
	_nNewLength	: INT;
END_VAR
Inject := _this;

IF sToInject = '' THEN
	RETURN;
END_IF

IF nPosition = 0 THEN
	RETURN;
END_IF

IF nPosition > _nLength THEN
	RETURN;
END_IF

_nNewLength := Tc2_Standard.LEN(sToInject) + _nLength;
IF _nNewLength > 255 THEN
	_nNewLength := 255;
END_IF

_sString := Tc2_Standard.INSERT(_sString, sToInject, nPosition);
_nLength := _nNewLength;
END_METHOD

// Checks if the current string is empty.
METHOD IsEmpty : BOOL
VAR_INPUT
END_VAR
IsEmpty := _nLength = 0;
END_METHOD

// Returns the current length of the string.
// The length of the string is stored as a separate variable (_nLength) 
// and reflects the actual length of the content.
// Unlike Tc2_Standard.LEN(), which counts up to the first null character, 
// this method directly returns the stored length.
METHOD Length : INT
VAR_INPUT
END_VAR
Length := _nLength;
END_METHOD

// Prepends the specified string to the current string.
// Truncates if the total length exceeds 255 characters.
METHOD Prepend : I_Strb
VAR_INPUT
    sToAdd : Str; // String to prepend
END_VAR
VAR
	_nNewLength	: INT;
END_VAR
Prepend := _this;

IF sToAdd = '' THEN
	RETURN;
END_IF

_nNewLength := Tc2_Standard.LEN(sToAdd) + _nLength;
IF _nNewLength > 255 THEN
	_nNewLength := 255;
END_IF

_sString := Tc2_Standard.CONCAT(sToAdd, _sString);
_nLength := _nNewLength;
END_METHOD

// Returns the current string value.
METHOD Read : Str
VAR_INPUT
END_VAR
Read := _sString;
END_METHOD

// Removes a substring of specified length starting at a given position.
METHOD Remove : I_Strb
VAR_INPUT
    nLength : INT;    // Length of the substring to remove
    nPosition : INT;  // Starting position of the substring to remove
END_VAR

VAR
	_nPosition	: INT;
END_VAR
Remove := _this;

IF nPosition = 0 THEN
	RETURN;
END_IF

IF nPosition > _nLength THEN
	RETURN;
END_IF

IF nLength = 0 THEN
	RETURN;
END_IF

IF nLength + nPosition > _nLength THEN
	nLength := _nLength - nPosition + 1;
END_IF

_sString := Tc2_Standard.DELETE(_sString, nLength, nPosition);
_nLength := _nLength - nLength;
END_METHOD

// Sets the current string to a new value.
METHOD Set : I_Strb
VAR_INPUT
    sLiteral : Str; // New string value
END_VAR
Set 		:= _this;

_sString 	:= sLiteral;
_nLength	:= Tc2_Standard.LEN(sLiteral);
END_METHOD

// Extracts a substring starting from a given position with a specified length.
METHOD Slice : I_Strb
VAR_INPUT
    nLength : INT;   // Length of the slice
    nPosition : INT; // Starting position of the slice
END_VAR
VAR_OUTPUT
    sSlice : Strb;   // The sliced string
END_VAR
Slice := _this;

IF nPosition = 0 THEN
	RETURN;
END_IF

IF nLength = 0 THEN
	RETURN;
END_IF

sSlice.Set(Tc2_Standard.MID(_sString, nLength, nPosition));
END_METHOD

// Splits the string into two parts at the specified position.
METHOD Split : I_Strb
VAR_INPUT
    nPosition : INT; // Position to split the string
END_VAR
VAR_OUTPUT
    sLeft : Strb;    // Left part of the split
    sRight : Strb;   // Right part of the split
END_VAR
Split := _this;

IF nPosition = 0 THEN
	RETURN;
END_IF

sLeft.Set(Tc2_Standard.LEFT(_sString, nPosition));
sRight.Set(Tc2_Standard.RIGHT(_sString, _nLength - nPosition));
END_METHOD

END_FUNCTION_BLOCK

// Strings/Strf/Strf
// The Strf provides utilities for string formatting.
PROGRAM Strf

// Formats a string using Tc2_Utilities.FB_FormatString with a single argument.
METHOD Fmt : Str
VAR_INPUT
	sFormat			: Str; // Format, check format specification on Beckhoff infosys.
	tcArg			: Tc2_Utilities.T_Arg;
END_VAR
VAR
	_fmt			: Tc2_Utilities.FB_FormatString;
END_VAR
_fmt(sFormat := sFormat, arg1 := tcArg, sOut => Fmt);
END_METHOD

// Adds left and/or right padding to a string with a specified fill character.
// Returns the padded string.
METHOD Padding : Str
VAR_INPUT
    sValue       : Str;  // The original string
    nLeftPadding : USINT := 0; // Number of padding characters to add to the left
    nRightPadding: USINT := 0; // Number of padding characters to add to the right
    sFillChar    : Ch := ' ';  // Character used for padding
END_VAR
VAR
	_nLen		: INT := Tc2_Standard.LEN(sValue);
	_nLeftMiss	: INT;
	_nRightMiss	: INT;	

	i			: INT;
END_VAR
_nLeftMiss := nLeftPadding - _nLen;
_nRightMiss := nRightPadding - _nLen;

IF _nLeftMiss > 0 THEN
	FOR i := 1 TO _nleftMiss DO
		sValue := Tc2_Standard.CONCAT(sFillChar, sValue);
	END_FOR	
END_IF

IF _nRightMiss > 0 THEN
	FOR i := 1 TO _nRightMiss DO
		sValue := Tc2_Standard.CONCAT(sFillChar, sValue);
	END_FOR	
END_IF

Padding := sValue;
END_METHOD

// Converts a TIME value to a human-readable string with specified minimum and maximum units.
// Returns the formatted time string.
METHOD SimpleTime : Str
VAR_INPUT
    tValue   : TIME;  // Time value to convert
    sMinUnit : Str := 'MS'; // Minimum unit (e.g., MS, S, M, H, D)
    sMaxUnit : Str := 'S';  // Maximum unit (e.g., MS, S, M, H, D)
END_VAR
VAR
	_nMinUnit	: USINT;
	_nMaxUnit	: USINT;
	_sValues	: ARRAY[1..5] OF Strb;
	_nValues	: ARRAY[1..5] OF UINT;
	_sUnits   	: ARRAY[1..5] OF STRING := ['MS', 'S', 'M', 'H', 'D'];
	_stTime		: Tc2_Utilities.OTSTRUCT;
	_i			: USINT;
	_strb		: Strb;
END_VAR
FOR _i := 1 TO 5 DO
	IF _sUnits[_i] = sMinUnit THEN
		_nMinUnit := _i;
	END_IF
	IF _sUnits[_i] = sMaxUnit THEN
		_nMaxUnit := _i;
	END_IF
END_FOR

IF _nMaxUnit = 0 THEN
	RETURN;
END_IF

IF _nMinUnit = 0 THEN
	RETURN;
END_IF

IF _nMinUnit > _nMaxUnit THEN
	RETURN;
END_IF

_stTime := Tc2_Utilities.TIME_TO_OTSTRUCT(tValue);
_stTime.wDay := _stTime.wWeek * 7 + _stTime.wDay;

_nValues[1] := WORD_TO_UINT(_stTime.wMilliseconds);
_nValues[2] := WORD_TO_UINT(_stTime.wSecond);
_nValues[3] := WORD_TO_UINT(_stTime.wMinute);
_nValues[4] := WORD_TO_UINT(_stTime.wHour);
_nValues[5] := WORD_TO_UINT(_stTime.wDay);

_sValues[1].Set(Strf.Padding(UINT_TO_STRING(_nValues[1]), 3, 0, '0')).Append('ms');
_sValues[2].Set(Strf.Padding(UINT_TO_STRING(_nValues[2]), 2, 0, '0')).Append('s');
_sValues[3].Set(Strf.Padding(UINT_TO_STRING(_nValues[3]), 2, 0, '0')).Append('m');
_sValues[4].Set(Strf.Padding(UINT_TO_STRING(_nValues[4]), 2, 0, '0')).Append('h');
_sValues[5].Set(Strf.Padding(UINT_TO_STRING(_nValues[5]), 3, 0, '0')).Append('d');

IF _nMaxUnit < 5 THEN
    FOR _i := 5 TO _nMaxUnit + 1 BY -1 DO
        IF _nValues[_i] <> 0 THEN
            _strb.Append(_sValues[_i].Read()).Append(' ');
        END_IF
    END_FOR
END_IF

FOR _i := _nMaxUnit TO _nMinUnit BY -1 DO
    _strb.Append(_sValues[_i].Read()).Append(' ');
END_FOR

SimpleTime := _strb.Read();
END_METHOD

END_PROGRAM

// Tags/Casts/IArgToITag
(*
Casts I_Arg as I_Tag.
Returns:
- Ok - Success,
- Err.InvRef - Invalid reference,
- Err.Itf0 - Invalid interface,
- Err.NoMatch - Cast failed
*)
FUNCTION IArgToITag : Result
VAR_INPUT
	iIn		: I_Arg;
	iOut	: REFERENCE TO I_Tag;
END_VAR

IF NOT __ISVALIDREF(iOut) THEN
	IArgToITag := Err.InvRef;
	RETURN;
END_IF

IF iIn = 0 THEN
	IArgToITag := Err.Itf0;
	RETURN;
END_IF

IF __QUERYINTERFACE(iIn, iOut) THEN
	IArgToITag := Ok;
ELSE
	IArgToITag := Err.NoMatch;
END_IF

END_FUNCTION

// Tags/Casts/ICompToITag
(*
Casts I_Component as I_Tag.
Returns:
- Ok - Success,
- Err.InvRef - Invalid reference,
- Err.Itf0 - Invalid interface,
- Err.NoMatch - Cast failed
*)
FUNCTION ICompToITag : Result
VAR_INPUT
	iIn		: I_Component;
	iOut	: REFERENCE TO I_Tag;
END_VAR

IF NOT __ISVALIDREF(iOut) THEN
	ICompToITag := Err.InvRef;
	RETURN;
END_IF

IF iIn = 0 THEN
	ICompToITag := Err.Itf0;
	RETURN;
END_IF

IF __QUERYINTERFACE(iIn, iOut) THEN
	ICompToITag := Ok;
ELSE
	ICompToITag := Err.NoMatch;
END_IF

END_FUNCTION

// Tags/Casts/ICompToITagged
(*
Casts I_Component as I_Tagged.
Returns:
- Ok - Success,
- Err.InvRef - Invalid reference,
- Err.Itf0 - Invalid interface,
- Err.NoMatch - Cast failed
*)
FUNCTION ICompToITagged : Result
VAR_INPUT
	iIn		: I_Component;
	iOut	: REFERENCE TO I_Tagged;
END_VAR

IF NOT __ISVALIDREF(iOut) THEN
	ICompToITagged := Err.InvRef;
	RETURN;
END_IF

IF iIn = 0 THEN
	ICompToITagged := Err.Itf0;
	RETURN;
END_IF

IF __QUERYINTERFACE(iIn, iOut) THEN
	ICompToITagged := Ok;
ELSE
	ICompToITagged := Err.NoMatch;
END_IF

END_FUNCTION

// Tags/Helpers/GetTag
(*
Searches an `I_Entity` for a `I_Tag` component matching provided id pattern.
Result:
- Ok - Returns iTag.
- Err.NotFound - Returns null.
- Err.InvRef - Provided reference is invalid.
- Err.Itf0 - Returns null, incorrect interface.
*)
FUNCTION GetTag : Result
VAR_INPUT
	iEntity		: I_Entity;
	sIdPattern	: Str;
	iOut		: REFERENCE TO I_Tag;
END_VAR
VAR
	i			: Iter(1);
	_iComp		: I_FatComponent;
	cmp			: TagCmp;
END_VAR

IF iEntity = 0 THEN
	GetTag := Err.Itf0;
	RETURN;
END_IF

IF NOT __ISVALIDREF(iOut) THEN
	GetTag := Err.InvRef;
	RETURN;
END_IF

WHILE IsOk(iEntity.Get(i.Next(), _iComp)) DO
	IF IsOk(ICompToITag(_iComp.Raw, iOut)) THEN
		IF cmp.Set(iOut).MatchWcdId(sIdPattern).IsTrue() THEN
			GetTag := Ok;
			RETURN;
		ELSE
			iOut := 0;
		END_IF
	END_IF
END_WHILE

GetTag := Err.NotFound;

END_FUNCTION

// Tags/Helpers/GetTagOption
(*
Searches an `I_Entity` for a `I_Tag` component with provided `Option` value.
Result:
- Ok - Returns iTag.
- Err.NotFound - Returns null.
- Err.InvRef - Provided reference is invalid.
- Err.Itf0 - Returns null, incorrect interface.
*)
FUNCTION GetTagOption : Result
VAR_INPUT
	iEntity		: I_Entity;
	sOption		: Str;
	iOut		: REFERENCE TO I_Tag;
END_VAR
VAR
	i			: Iter(1);
	_iComp		: I_FatComponent;
END_VAR

IF iEntity = 0 THEN
	GetTagOption := Err.Itf0;
	RETURN;
END_IF

IF NOT __ISVALIDREF(iOut) THEN
	GetTagOption := Err.InvRef;
	RETURN;
END_IF

WHILE IsOk(iEntity.Get(i.Next(), _iComp)) DO
	IF IsOk(ICompToITag(_iComp.Raw, iOut)) THEN
		IF iOut.Option = sOption THEN
			GetTagOption := Ok;
			RETURN;
		ELSE
			iOut := 0;
		END_IF
	END_IF
END_WHILE

GetTagOption := Err.NotFound;

END_FUNCTION

// Tags/Helpers/HasTag
(*
Searches an `I_Entity` for a `I_Tag` component matching provided id pattern.
Result:
- Ok
- Err.NotFound - Returns null.
- Err.Itf0 - Returns null, incorrect interface.
*)
FUNCTION HasTag : Result
VAR_INPUT
	iEntity		: I_Entity;
	sIdPattern	: Str;
END_VAR
VAR
	i			: Iter(1);
	_iComp		: I_FatComponent;
	_iTag		: I_Tag;
	cmp			: TagCmp;
END_VAR

IF iEntity = 0 THEN
	HasTag := Err.Itf0;
	RETURN;
END_IF

WHILE IsOk(iEntity.Get(i.Next(), _iComp)) DO
	IF IsOk(ICompToITag(_iComp.Raw, _iTag)) THEN
		IF cmp.Set(_iTag).MatchWcdId(sIdPattern).IsTrue() THEN
			HasTag := Ok;
			RETURN;
		END_IF
	END_IF
END_WHILE

HasTag := Err.NotFound;

END_FUNCTION

// Tags/Helpers/HasTagOption
(*
Searches an `I_Entity` for a `I_Tag` component with provided `Option` value.
Result:
- Ok
- Err.NotFound - Returns null.
- Err.Itf0 - Returns null, incorrect interface.
*)
FUNCTION HasTagOption : Result
VAR_INPUT
	iEntity		: I_Entity;
	sOption		: Str;
END_VAR
VAR
	i			: Iter(1);
	_iComp		: I_FatComponent;
	_iTag		: I_Tag;
END_VAR

IF iEntity = 0 THEN
	HasTagOption := Err.Itf0;
	RETURN;
END_IF

WHILE IsOk(iEntity.Get(i.Next(), _iComp)) DO
	IF IsOk(ICompToITag(_iComp.Raw, _iTag)) THEN
		IF _iTag.Option = sOption THEN
			HasTagOption := Ok;
			RETURN;
		END_IF
	END_IF
END_WHILE

HasTagOption := Err.NotFound;

END_FUNCTION
